ABB RobotStudio station: regno.210021601039.rspag

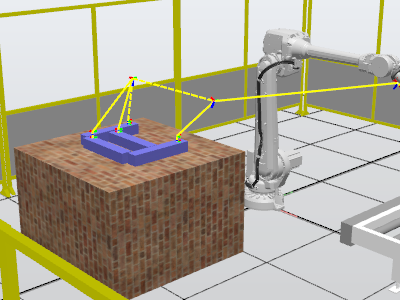
--- station ---
Station Aslam (saved by RobotStudio 23.2.10478.1)
Controller Controller1
  mechanical unit ROB_1: IRB4600_40_255_C_01, 6 joints, base frame (0, 0, 0) mm
Layout (positions relative to the parent item):
  - IRB4600_40_255_C_01 [mechanism, from %ABB.RobotStudio.Models.IRB4600%\IRB4600_40_255_C_G_01.rslib] at (0, 0, 0) mm; joint values [0, 0, 0, 0, 0.5236, 0] (rad or m)
  - Smart_Gripper_Servo_One_Vacuum [mechanism, from %ABB.RobotStudio.Models.SmartGripper%\ABB_Smart_Gripper_Servo_One_Vacuum.rslib] at (1561.91, 0, 1697.5) mm, rotated rx 180 ry 60 rz 180 deg; joint values [0] (rad or m)
  - 950_4000_h2 [part, from %ABB.RobotStudio.Models.Conveyors%\Conveyor 950 4000 h2.rslib] at (1600, -500, 0) mm
  - Part_1 [part] at (-800, -2500, 0) mm, size 1500 x 1500 x 1000 mm
  - conveyor [smart component]
      signals: DI di_IP, DO Di_op
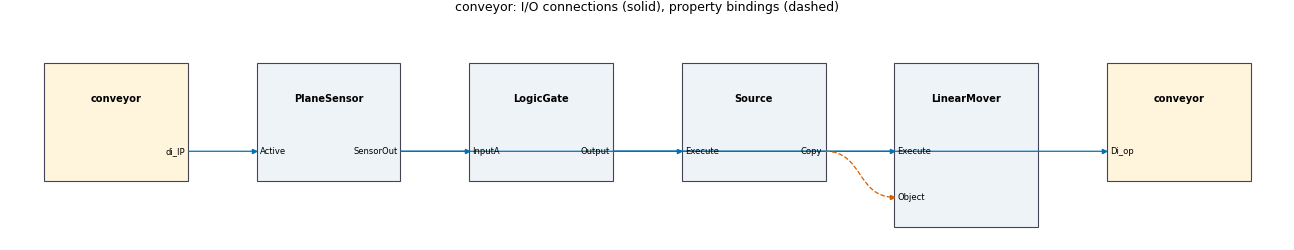
      connections:
        conveyor.di_IP -> PlaneSensor.Active
        PlaneSensor.SensorOut -> conveyor.Di_op
        PlaneSensor.SensorOut -> LogicGate.InputA
        LogicGate.Output -> Source.Execute
        LogicGate.Output -> LinearMover.Execute
        Source.Copy => LinearMover.Object
    - PlaneSensor [smart component, from Components\PlaneSensor.rslib] at (1999, -400, 435) mm
        properties: Origin=[0 0 0]; Axis1=[0 0 0.1]; Axis2=[0 0.7 0]; Tag=(none); SensedPart=Part_3_21
      - _sensorPart_ [part], size 0 x 700 x 100 mm
    - Source [smart component, from Components\Source.rslib]
        properties: Source=Part_3; Copy=Part_3_21; Parent=(none); Position=[0 0 0]; Orientation=[0 0 0]; Transient=false; PhysicsBehavior=-1
    - LogicGate [smart component, from Components\LogicGate.rslib]
        properties: Operator=NOT; Delay=0
    - SimulationEvents [smart component, from Components\SimulationEvents.rslib]
    - LinearMover [smart component, from Components\LinearMover.rslib]
        properties: Object=Part_3_21; Direction=[-4 0 0]; Speed=1; Reference=Global; ReferenceObject=(none)
  - sc_gripper [smart component]
      signals: DI di_ip, DO di_op
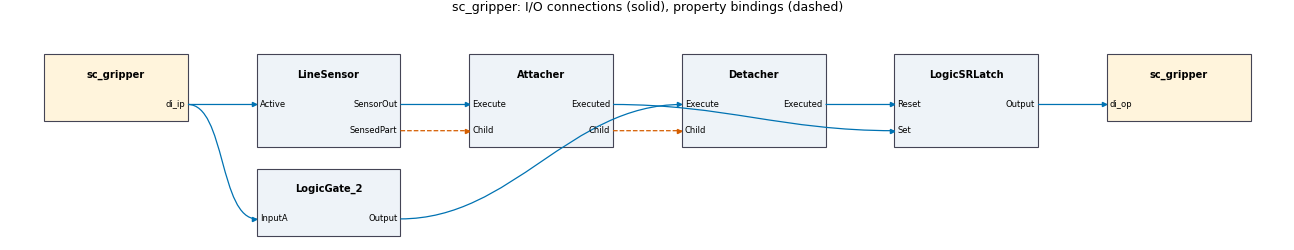
      connections:
        sc_gripper.di_ip -> LineSensor.Active
        sc_gripper.di_ip -> LogicGate_2.InputA
        LineSensor.SensorOut -> Attacher.Execute
        LogicGate_2.Output -> Detacher.Execute
        Detacher.Executed -> LogicSRLatch.Reset
        Attacher.Executed -> LogicSRLatch.Set
        LogicSRLatch.Output -> sc_gripper.di_op
        LineSensor.SensedPart => Attacher.Child
        Attacher.Child => Detacher.Child
    - LineSensor [smart component, from Components\LineSensor.rslib] at (1569.39, 18.5, 1635.45) mm, rotated rx 180 ry -30 rz 180 deg
        properties: Start=[0 0 0]; End=[0 0 0.02]; Length=0.02; Radius=0.0005; Tag=(none); SensedPart=Part_3_20; SensedPoint=[0.305250396728516 -1.47408911132812 1.09926806640625]
      - _sensorPart_ [part], size 1 x 1 x 20 mm
    - LogicGate_2 [smart component, from Components\LogicGate.rslib]
        properties: Operator=NOT; Delay=0
    - Attacher [smart component, from Components\Attacher.rslib]
        properties: Parent=Smart_Gripper_Servo_One_Vacuum; Flange=1; Child=Part_3_20; Mount=false; Offset=[0 0 0]; Orientation=[0 0 0]
    - Detacher [smart component, from Components\Detacher.rslib]
        properties: Child=Part_3_20; KeepPosition=true
    - LogicSRLatch [smart component, from Components\LogicSRLatch.rslib]
  - Part_3 [part], size 600 x 100 x 100 mm
  - Fence_2500 [graphiccomponentgroup, from Equipment\Fence_2500.rslib] at (-2100.49, -4439.5, 0) mm
    - Body 1 [part, from Equipment\Fence_2500.rslib]
    - Body 2 [part, from Equipment\Fence_2500.rslib]
  - Fence_2500_2 [graphiccomponentgroup, from Equipment\Fence_2500.rslib] at (7907.06, -1867.5, 0) mm
    - Body 1 [part, from Equipment\Fence_2500.rslib]
    - Body 2 [part, from Equipment\Fence_2500.rslib]
  - Fence_2500_3 [graphiccomponentgroup, from Equipment\Fence_2500.rslib] at (-2089.16, 592.51, 0) mm
    - Body 1 [part, from Equipment\Fence_2500.rslib]
    - Body 2 [part, from Equipment\Fence_2500.rslib]
  - Fence_2500_4 [graphiccomponentgroup, from Equipment\Fence_2500.rslib] at (-2003.24, 3066.49, 0) mm, rotated rx 0 ry 0 rz -88.91 deg
    - Body 1 [part, from Equipment\Fence_2500.rslib]
    - Body 2 [part, from Equipment\Fence_2500.rslib]
  - Fence_2500_5 [graphiccomponentgroup, from Equipment\Fence_2500.rslib] at (500.31, 3070.54, 0) mm, rotated rx 0 ry 0 rz -89.71 deg
    - Body 1 [part, from Equipment\Fence_2500.rslib]
    - Body 2 [part, from Equipment\Fence_2500.rslib]
  - Fence_2500_6 [graphiccomponentgroup, from Equipment\Fence_2500.rslib] at (3010.78, 3112.98, 0) mm, rotated rx 0 ry 0 rz -89.71 deg
    - Body 1 [part, from Equipment\Fence_2500.rslib]
    - Body 2 [part, from Equipment\Fence_2500.rslib]
  - Fence_2500_7 [graphiccomponentgroup, from Equipment\Fence_2500.rslib] at (5530.17, 3122.93, 0) mm, rotated rx 0 ry 0 rz -89.71 deg
    - Body 1 [part, from Equipment\Fence_2500.rslib]
    - Body 2 [part, from Equipment\Fence_2500.rslib]
  - Fence_2500_8 [graphiccomponentgroup, from Equipment\Fence_2500.rslib] at (-2202.71, -4426.51, 0) mm, rotated rx 0 ry 0 rz -89.71 deg
    - Body 1 [part, from Equipment\Fence_2500.rslib]
    - Body 2 [part, from Equipment\Fence_2500.rslib]
  - Fence_2500_9 [graphiccomponentgroup, from Equipment\Fence_2500.rslib] at (323.09, -4426.65, 0) mm, rotated rx 0 ry 0 rz -89.71 deg
    - Body 1 [part, from Equipment\Fence_2500.rslib]
    - Body 2 [part, from Equipment\Fence_2500.rslib]
  - Fence_2500_10 [graphiccomponentgroup, from Equipment\Fence_2500.rslib] at (5359.98, -4393.32, 5.38) mm, rotated rx 0 ry 0 rz -89.71 deg
    - Body 1 [part, from Equipment\Fence_2500.rslib]
    - Body 2 [part, from Equipment\Fence_2500.rslib]
  - Fence_2500_11 [graphiccomponentgroup, from Equipment\Fence_2500.rslib] at (2827.43, -4425.85, 5.38) mm, rotated rx 0 ry 0 rz -89.71 deg
    - Body 1 [part, from Equipment\Fence_2500.rslib]
    - Body 2 [part, from Equipment\Fence_2500.rslib]
  - Fence_2500_12 [graphiccomponentgroup, from Equipment\Fence_2500.rslib] at (7899.47, -4400.73, 0) mm
    - Body 1 [part, from Equipment\Fence_2500.rslib]
    - Body 2 [part, from Equipment\Fence_2500.rslib]
  - Fence_2500_14 [graphiccomponentgroup, from Equipment\Fence_2500.rslib] at (-2089.16, -1922.77, 22.33) mm
    - Body 1 [part, from Equipment\Fence_2500.rslib]
    - Body 2 [part, from Equipment\Fence_2500.rslib]
  - Gate [graphiccomponentgroup, from Equipment\Fence_Gate.rslib] at (7969.77, 744.51, 0) mm
    - Body 1 [part, from Equipment\Fence_Gate.rslib]
    - Body 2 [part, from Equipment\Fence_Gate.rslib]
    - Body 3 [part, from Equipment\Fence_Gate.rslib]
  - Fence_740 [graphiccomponentgroup, from Equipment\Fence_740.rslib] at (7986.63, 2332.89, 0) mm
    - Body 1 [part, from Equipment\Fence_740.rslib]
    - Body 2 [part, from Equipment\Fence_740.rslib]
  - Part_3_17 [part] at (-5363.03, -1931.8, 541.89) mm, rotated rx 0 ry -0.05 rz 0 deg, size 600 x 100 x 100 mm
  - Part_3_18 [part] at (-5360.93, -1650, 539.31) mm, rotated rx 0 ry -0.05 rz 0 deg, size 600 x 100 x 100 mm
  - Part_3_19 [part] at (-413.78, 3611.12, 572.22) mm, rotated rx 0 ry 0.2 rz -89.45 deg, size 600 x 100 x 100 mm
  - Part_3_20 [part] at (306.1, 3612.36, 541.18) mm, rotated rx 0 ry -0.09 rz -89.45 deg, size 600 x 100 x 100 mm
  - Part_3_21 [part] at (-3024, 0, 0) mm, size 600 x 100 x 100 mm
Attachment: Smart_Gripper_Servo_One_Vacuum is attached to IRB4600_40_255_C_01 / Link6
Attachment: LineSensor is attached to Smart_Gripper_Servo_One_Vacuum / DownFinger
Station logic (signal -> signal, property => property):
  Controller1.di_outp -> conveyor.di_IP
  Controller1.out -> sc_gripper.di_ip
  conveyor.Di_op -> Controller1.start

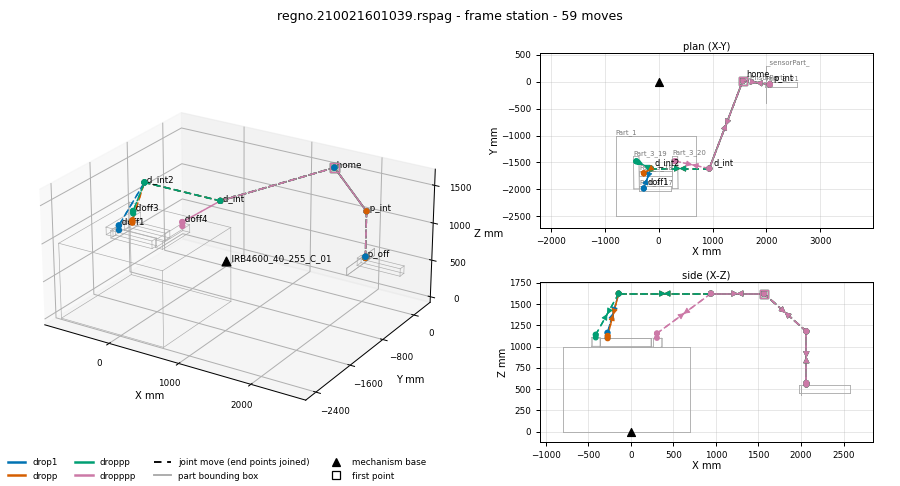
[picture p0: tool path of regno.210021601039.rspag in frame station, 59 of 59 moves have a stored position in this frame; points joined in program order, loops and branches not executed]
--- Controller Data/Controller1/RAPID/TASK1/PROGMOD/CalibData.mod ---
MODULE CalibData
    PERS tooldata Servo:=[TRUE,[[0,0,84],[1,0,0,0]],[0.226,[8.9,12.3,48.7],[1,0,0,0],0.00021,0.00024,0.00009]];
    PERS tooldata VaccumOne:=[TRUE,[[63.5,18.5,37.5],[0.707106781,0,0.707106781,0]],[0.226,[8.9,12.3,48.7],[1,0,0,0],0.00021,0.00024,0.00009]];
ENDMODULE

--- Controller Data/Controller1/RAPID/TASK1/PROGMOD/Module1.mod ---
MODULE Module1
        CONST robtarget home:=[[1562.639382153,18.5,1623.75738686],[0.258819045,0,-0.965925826,0],[-1,0,-1,0],[9E+09,9E+09,9E+09,9E+09,9E+09,9E+09]];
    CONST robtarget p_int:=[[2063.172095275,-50.000005327,1179.24592598],[0.258819026,-0.000000016,-0.965925831,0.000000083],[-1,-4,3,0],[9E+09,9E+09,9E+09,9E+09,9E+09,9E+09]];
    CONST robtarget p_off:=[[2063.172096002,-50.000028315,570.499577423],[0.015201551,-0.000000059,-0.99988445,0.00000017],[-1,-3,2,0],[9E+09,9E+09,9E+09,9E+09,9E+09,9E+09]];
    CONST robtarget pick:=[[2063.172094301,-50.000051782,552.69067907],[0.015201544,-0.000000044,-0.99988445,0.000000279],[-1,-3,2,0],[9E+09,9E+09,9E+09,9E+09,9E+09,9E+09]];
    CONST robtarget d_int:=[[940.228552583,-1612.069048412,1623.756948723],[0.258819034,0.000000012,-0.965925829,-0.00000002],[-1,0,-1,0],[9E+09,9E+09,9E+09,9E+09,9E+09,9E+09]];
    CONST robtarget d_int2:=[[-144.835901472,-1612.069029255,1623.756967463],[0.014740524,-0.000000036,-0.999891353,-0.000000019],[-2,0,-2,0],[9E+09,9E+09,9E+09,9E+09,9E+09,9E+09]];
    CONST robtarget drop:=[[-276.361767602,-1981.811058938,1101.884003045],[0.014740521,-0.000000099,-0.999891353,-0.000000006],[-2,0,-2,0],[9E+09,9E+09,9E+09,9E+09,9E+09,9E+09]];
    CONST robtarget drop2:=[[-274.268306528,-1700.000070232,1096.688942945],[0.014740539,-0.000000063,-0.999891352,0.000000035],[-2,0,-2,0],[9E+09,9E+09,9E+09,9E+09,9E+09,9E+09]];
    CONST robtarget d_int2s3:=[[-144.835846566,-1612.069030946,1623.756982975],[0.00040913,-0.703683907,-0.710513017,-0.000210601],[-2,1,-2,0],[9E+09,9E+09,9E+09,9E+09,9E+09,9E+09]];
    CONST robtarget drop3:=[[-414.630501937,-1478.227007764,1106.829966049],[0.012047983,-0.703580919,-0.710412296,-0.011962693],[-2,1,-2,0],[9E+09,9E+09,9E+09,9E+09,9E+09,9E+09]];
    CONST robtarget drop4:=[[305.251281504,-1474.166996213,1101.958917838],[0.010238324,-0.703609606,-0.710440698,-0.01013481],[-1,2,-3,0],[9E+09,9E+09,9E+09,9E+09,9E+09,9E+09]];
    CONST robtarget doff1:=[[-276.36176126,-1981.811048156,1163.043031401],[0.014740495,-0.0000001,-0.999891353,0.000000001],[-2,0,-2,0],[9E+09,9E+09,9E+09,9E+09,9E+09,9E+09]];
    CONST robtarget doff2:=[[-274.268301083,-1700.000061117,1126.373987512],[0.014740524,-0.000000072,-0.999891353,0.000000033],[-2,0,-2,0],[9E+09,9E+09,9E+09,9E+09,9E+09,9E+09]];
    CONST robtarget doff3:=[[-414.630504406,-1478.227029584,1139.901944465],[0.012048007,-0.7035809,-0.710412314,-0.01196268],[-2,1,-2,0],[9E+09,9E+09,9E+09,9E+09,9E+09,9E+09]];
    CONST robtarget doff4:=[[305.251147751,-1474.16703993,1154.976935412],[0.010237777,-0.703609816,-0.710440486,-0.010135552],[-1,2,-3,0],[9E+09,9E+09,9E+09,9E+09,9E+09,9E+09]];
    CONST robtarget Target_10:=[[1562.639382153,18.5,1623.75738686],[0.258819045,0,-0.965925826,0],[-1,0,-1,0],[9E+09,9E+09,9E+09,9E+09,9E+09,9E+09]];
!***********************************************************
    !
    ! Module:  Module1
    !
    ! Description:
    !   <Insert description here>
    !
    ! Author: shahu
    !
    ! Version: 1.0
    !
    !***********************************************************


    !***********************************************************
    !
    ! Procedure main
    !
    !   This is the entry point of your program
    !
    !***********************************************************
    PROC main()
        !Add your code here
    ENDPROC
    PROC drop1()
        MoveJ home,v1000,fine,VaccumOne\WObj:=wobj0;
        MoveJ p_int,v1000,fine,VaccumOne\WObj:=wobj0;
        MoveJ p_off,v1000,fine,VaccumOne\WObj:=wobj0;
        MoveJ pick,v1000,fine,VaccumOne\WObj:=wobj0;
        WaitTime 0.5;
        SetDO out,1;
        WaitTime 0.5;
        MoveJ p_off,v1000,fine,VaccumOne\WObj:=wobj0;
        MoveJ p_int,v1000,fine,VaccumOne\WObj:=wobj0;
        MoveJ home,v1000,fine,VaccumOne\WObj:=wobj0;
        MoveJ d_int,v1000,fine,VaccumOne\WObj:=wobj0;
        MoveJ d_int2,v1000,fine,VaccumOne\WObj:=wobj0;
        MoveJ doff1,v1000,fine,VaccumOne\WObj:=wobj0;
        MoveJ drop,v1000,fine,VaccumOne\WObj:=wobj0;
        WaitTime 0.5;
        SetDO out,0;
        WaitTime 0.5;
        MoveJ doff1,v1000,fine,VaccumOne\WObj:=wobj0;
        MoveJ d_int2,v1000,fine,VaccumOne\WObj:=wobj0;
        MoveJ d_int,v1000,fine,VaccumOne\WObj:=wobj0;
        MoveJ home,v1000,fine,VaccumOne\WObj:=wobj0;
    ENDPROC
    PROC dropp()
        MoveJ home,v1000,fine,VaccumOne\WObj:=wobj0;
        MoveJ p_int,v1000,fine,VaccumOne\WObj:=wobj0;
        MoveJ p_off,v1000,fine,VaccumOne\WObj:=wobj0;
        MoveJ pick,v1000,fine,VaccumOne\WObj:=wobj0;
        WaitTime 0.5;
        SetDO out,1;
        WaitTime 0.5;
        MoveJ p_off,v1000,fine,VaccumOne\WObj:=wobj0;
        MoveJ p_int,v1000,fine,VaccumOne\WObj:=wobj0;
        MoveJ home,v1000,fine,VaccumOne\WObj:=wobj0;
        MoveJ d_int,v1000,fine,VaccumOne\WObj:=wobj0;
        MoveJ d_int2,v1000,fine,VaccumOne\WObj:=wobj0;
        MoveJ doff2,v1000,fine,VaccumOne\WObj:=wobj0;
        MoveJ drop2,v1000,fine,VaccumOne\WObj:=wobj0;
        WaitTime 0.5;
        SetDO out,0;
        WaitTime 0.5;
        MoveJ doff2,v1000,fine,VaccumOne\WObj:=wobj0;
        MoveJ d_int2,v1000,fine,VaccumOne\WObj:=wobj0;
        MoveJ d_int,v1000,fine,VaccumOne\WObj:=wobj0;
        MoveJ home,v1000,fine,VaccumOne\WObj:=wobj0;
    ENDPROC
    PROC droppp()
        MoveJ home,v1000,fine,VaccumOne\WObj:=wobj0;
        MoveJ p_int,v1000,fine,VaccumOne\WObj:=wobj0;
        MoveJ p_off,v1000,fine,VaccumOne\WObj:=wobj0;
        MoveJ pick,v1000,fine,VaccumOne\WObj:=wobj0;
        WaitTime 0.5;
        SetDO out,1;
        WaitTime 0.5;
        MoveJ p_off,v1000,fine,VaccumOne\WObj:=wobj0;
        MoveJ p_int,v1000,fine,VaccumOne\WObj:=wobj0;
        MoveJ home,v1000,fine,VaccumOne\WObj:=wobj0;
        MoveJ d_int,v1000,fine,VaccumOne\WObj:=wobj0;
        MoveJ d_int2s3,v1000,fine,VaccumOne\WObj:=wobj0;
        MoveJ doff3,v1000,fine,VaccumOne\WObj:=wobj0;
        MoveJ drop3,v1000,fine,VaccumOne\WObj:=wobj0;
        WaitTime 0.5;
        SetDO out,0;
        WaitTime 0.5;
        MoveJ doff3,v1000,fine,VaccumOne\WObj:=wobj0;
        MoveJ d_int2s3,v1000,fine,VaccumOne\WObj:=wobj0;
        MoveJ d_int,v1000,fine,VaccumOne\WObj:=wobj0;
        MoveJ home,v1000,fine,VaccumOne\WObj:=wobj0;
        MoveJ home,v1000,fine,VaccumOne\WObj:=wobj0;
    ENDPROC
    PROC dropppp()
        MoveJ home,v1000,fine,VaccumOne\WObj:=wobj0;
        MoveJ p_int,v1000,fine,VaccumOne\WObj:=wobj0;
        MoveJ p_off,v1000,fine,VaccumOne\WObj:=wobj0;
        MoveJ pick,v1000,fine,VaccumOne\WObj:=wobj0;
        WaitTime 0.5;
        SetDO out,1;
        WaitTime 0.5;
        MoveJ p_off,v1000,fine,VaccumOne\WObj:=wobj0;
        MoveJ p_int,v1000,fine,VaccumOne\WObj:=wobj0;
        MoveJ home,v1000,fine,VaccumOne\WObj:=wobj0;
        MoveJ d_int,v1000,fine,VaccumOne\WObj:=wobj0;
        MoveJ doff4,v1000,fine,VaccumOne\WObj:=wobj0;
        MoveJ drop4,v1000,fine,VaccumOne\WObj:=wobj0;
        WaitTime 0.5;
        SetDO out,0;
        WaitTime 0.5;
        MoveJ doff4,v1000,fine,VaccumOne\WObj:=wobj0;
        MoveJ d_int,v1000,fine,VaccumOne\WObj:=wobj0;
        MoveJ home,v1000,fine,VaccumOne\WObj:=wobj0;
    ENDPROC
    PROC Path_10()

    ENDPROC
    PROC finalpath()
        WaitTime 3;
        drop1;
        dropp;
        droppp;
        dropppp;
    ENDPROC
ENDMODULE

--- Controller Data/Controller1/SYSPAR/EIO.cfg ---
EIO:CFG_1.0:6:1::
#
EIO_SIGNAL:

      -Name "start" -SignalType "DI" -Access "All"

      -Name "out" -SignalType "DO" -Access "All"

      -Name "di_outp" -SignalType "DO" -Access "All"
